// TIA Portal V18 export
DATA_BLOCK "SS1_710A1_8RTD_AI_Vars"   // DB11021
{ S7_Optimized_Access := 'FALSE' }
VERSION : 0.1
// stored: AutoNumber false, DBAccessibleFromOPCUA true, IsOnlyStoredInLoadMemory false, IsWriteProtectedInAS false
   VAR
      AI1 { S7_SetPoint := 'True'} : "UDT_RTDadv";   // Зовнішня температура (1.99)
      AI2 { S7_SetPoint := 'True'} : "UDT_RTDadv";   // AHU NF Темп. зв. теплоносія (2.57)
      AI3 { S7_SetPoint := 'True'} : "UDT_RTDadv";   // AHU NF Темп. припл. пов. (2.56)
      AI4 { S7_SetPoint := 'True'} : "UDT_RTDadv";   // AHU NF Кімнатна темп. (2.69)
      AI5 { S7_SetPoint := 'True'} : "UDT_RTDadv";   // HS Темп. под. теплоносія в колекторі (10.50)
      AI6 { S7_SetPoint := 'True'} : "UDT_RTDadv";   // Температура зв. теплоносія (8.66)
      AI7 { S7_SetPoint := 'True'} : "UDT_RTDadv";   // Темп. припл. пов. (8.68)
      AI8 { S7_SetPoint := 'True'} : "UDT_RTDadv";   // HS Темп. зв. теплоносія (10.92)
   END_VAR
BEGIN
   AI1.rValue := 26.03;
   AI1.rFilterSet := 0.0;
   AI1.rCalibration := 0.0;
   AI1.rDiv := 100.0;
   AI1.cFuncSystemID := 0;
   AI1.cFuncVar := 0;
   AI1.iReserv := 0;
   AI2.rValue := 3276.7;
   AI2.rFilterSet := 0.0;
   AI2.rCalibration := 0.0;
   AI2.rDiv := 10.0;
   AI2.cFuncSystemID := 2;
   AI2.cFuncVar := 0;
   AI2.iReserv := 0;
   AI3.rValue := 26.7;
   AI3.rFilterSet := 0.0;
   AI3.rCalibration := 0.0;
   AI3.rDiv := 100.0;
   AI3.cFuncSystemID := 16#01;
   AI3.cFuncVar := 16#04;
   AI3.iReserv := 0;
   AI4.rValue := 22.39;
   AI4.rFilterSet := 0.0;
   AI4.rCalibration := 0.0;
   AI4.rDiv := 100.0;
   AI4.cFuncSystemID := 16#03;
   AI4.cFuncVar := 16#04;
   AI4.iReserv := 0;
   AI5.rValue := 24.7;
   AI5.rFilterSet := 0.0;
   AI5.rCalibration := 0.0;
   AI5.rDiv := 10.0;
   AI5.cFuncSystemID := 16#0A;
   AI5.cFuncVar := 16#01;
   AI5.iReserv := 0;
   AI6.rValue := 61.78;
   AI6.rFilterSet := 0.0;
   AI6.rCalibration := 0.0;
   AI6.rDiv := 100.0;
   AI6.cFuncSystemID := 16#0E;
   AI6.cFuncVar := 16#01;
   AI6.iReserv := 0;
   AI7.rValue := 28.62;
   AI7.rFilterSet := 0.0;
   AI7.rCalibration := 0.0;
   AI7.rDiv := 100.0;
   AI7.cFuncSystemID := 16#0E;
   AI7.cFuncVar := 16#02;
   AI7.iReserv := 0;
   AI8.rValue := 21.31;
   AI8.rFilterSet := 0.0;
   AI8.rCalibration := 0.0;
   AI8.rDiv := 100.0;
   AI8.cFuncSystemID := 16#03;
   AI8.cFuncVar := 16#06;
   AI8.iReserv := 0;
END_DATA_BLOCK
